(* PLC project Unnamed, Unknown Unnamed 1 *)
(* stored: creationDateTime 2023-03-10T10:37:17, modificationDateTime 2023-03-15T15:56:42 *)

(* ISBN 978-3-8348-0266-8, Lernaufgabe 2.5 *)
FUNCTION_BLOCK Seven_Segment_Display
  VAR_INPUT
    IN0 : BOOL;
    IN1 : BOOL;
    IN2 : BOOL;
    IN3 : BOOL;
    IN4 : BOOL;
  END_VAR
  VAR_OUTPUT
    OUTa : BOOL;
    OUTb : BOOL;
    OUTc : BOOL;
    OUTd : BOOL;
    OUTe : BOOL;
    OUTf : BOOL;
    OUTg : BOOL;
  END_VAR

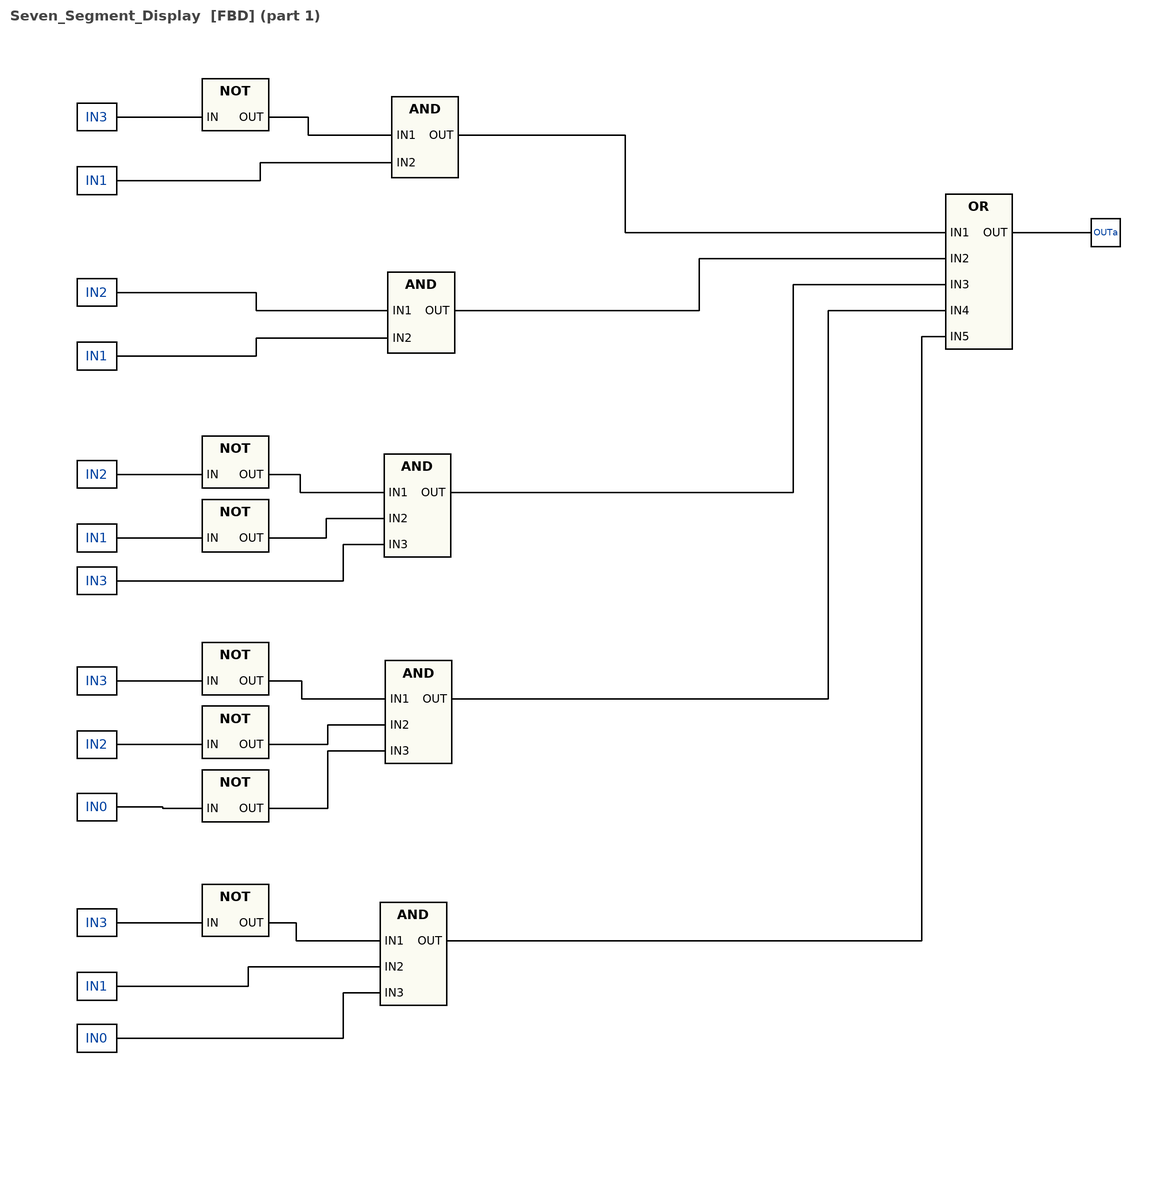
(* FBD diagram, written out as Structured Text *)
OUTa := NOT IN3 AND IN1 OR IN2 AND IN1 OR NOT IN2 AND NOT IN1 AND IN3 OR NOT IN3 AND NOT IN2 AND NOT IN0 OR NOT IN3 AND IN1 AND IN0;
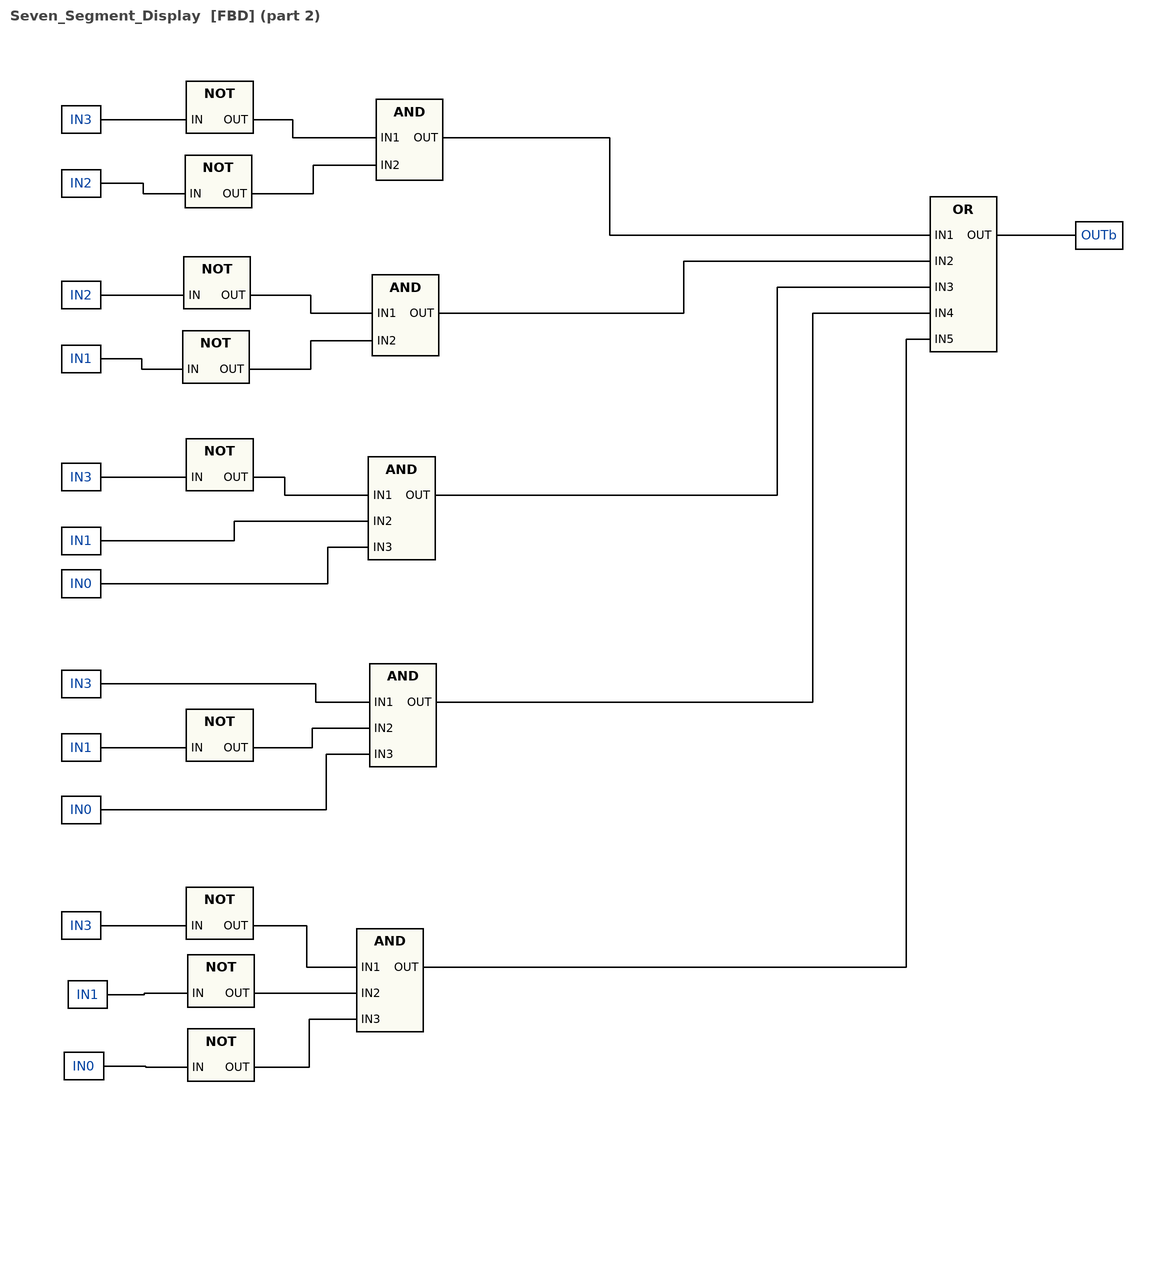
OUTb := NOT IN3 AND NOT IN2 OR NOT IN2 AND NOT IN1 OR NOT IN3 AND IN1 AND IN0 OR IN3 AND NOT IN1 AND IN0 OR NOT IN3 AND NOT IN1 AND NOT IN0;
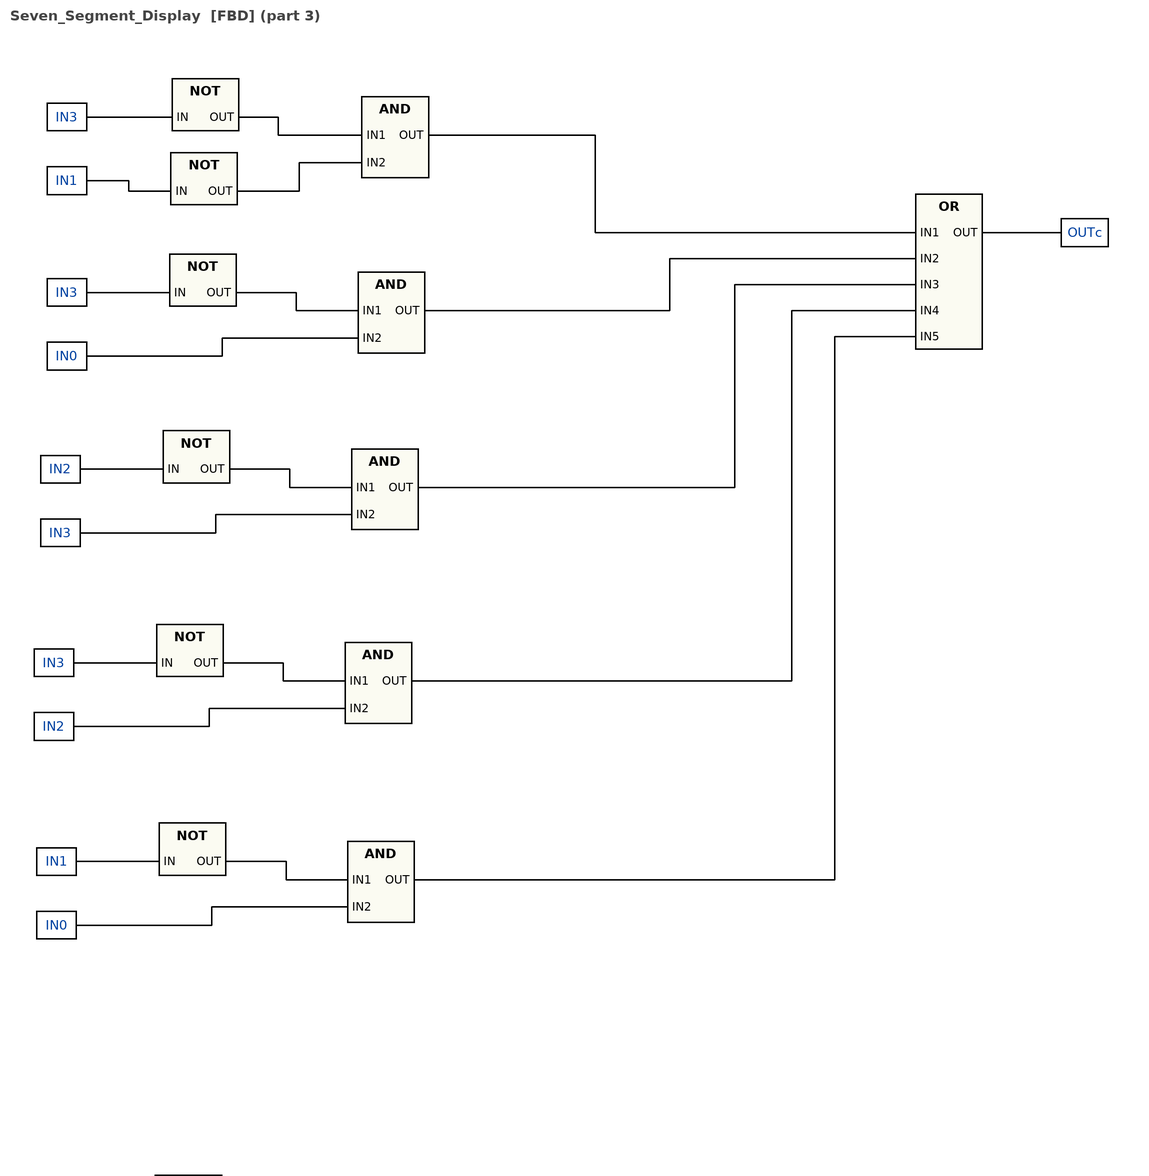
OUTc := NOT IN3 AND NOT IN1 OR NOT IN3 AND IN0 OR NOT IN2 AND IN3 OR NOT IN3 AND IN2 OR NOT IN1 AND IN0;
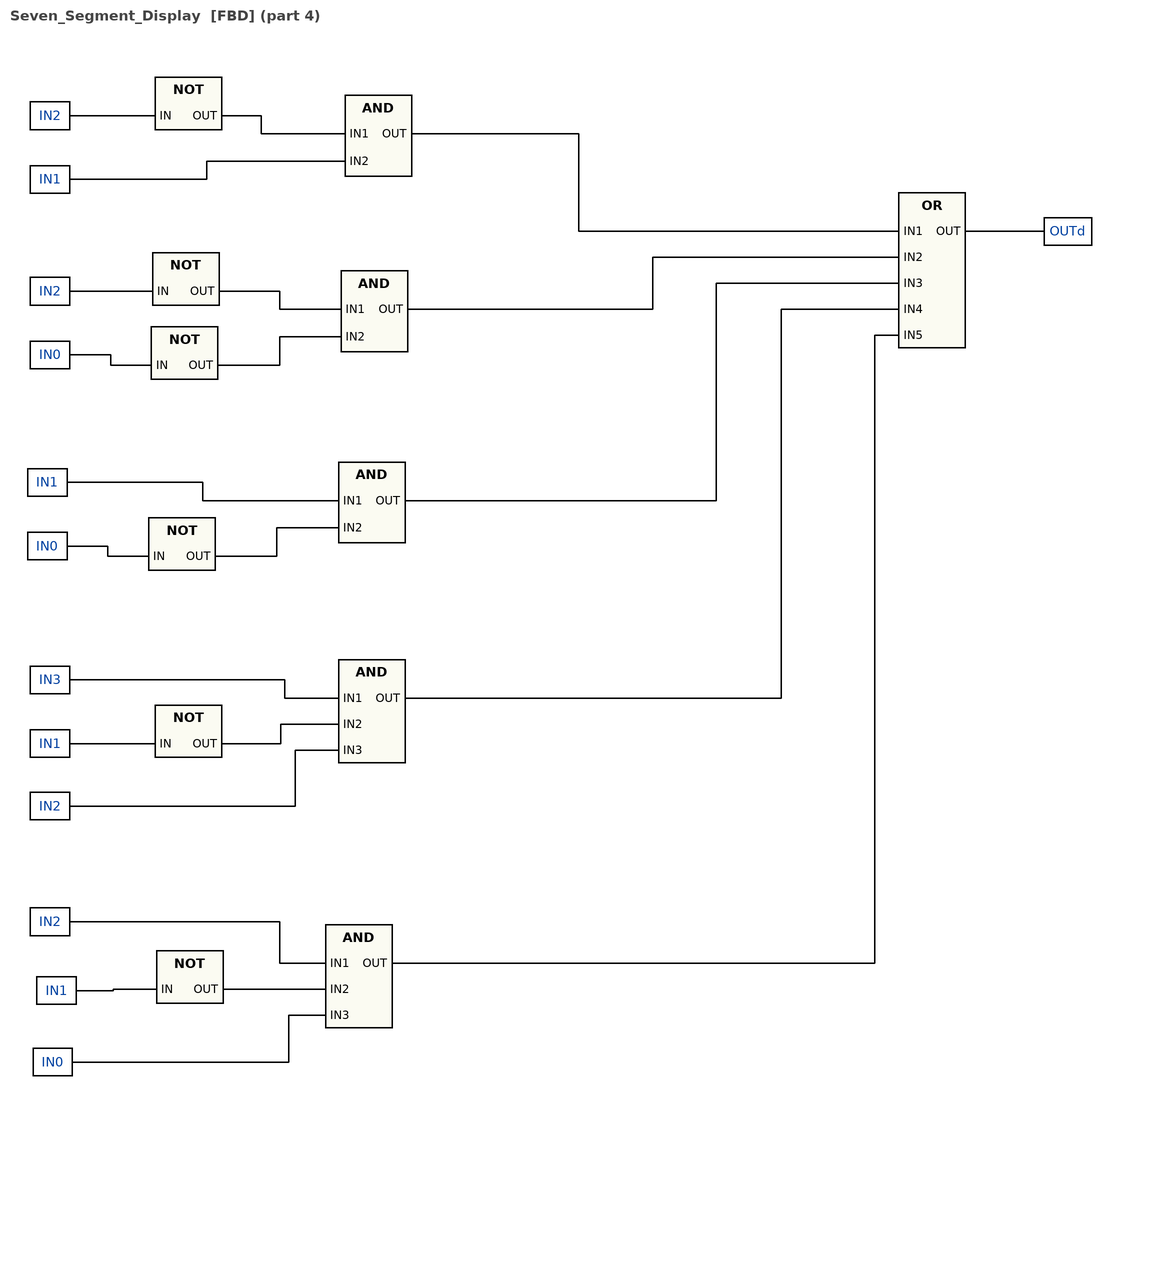
OUTd := NOT IN2 AND IN1 OR NOT IN2 AND NOT IN0 OR IN1 AND NOT IN0 OR IN3 AND NOT IN1 AND IN2 OR IN2 AND NOT IN1 AND IN0;
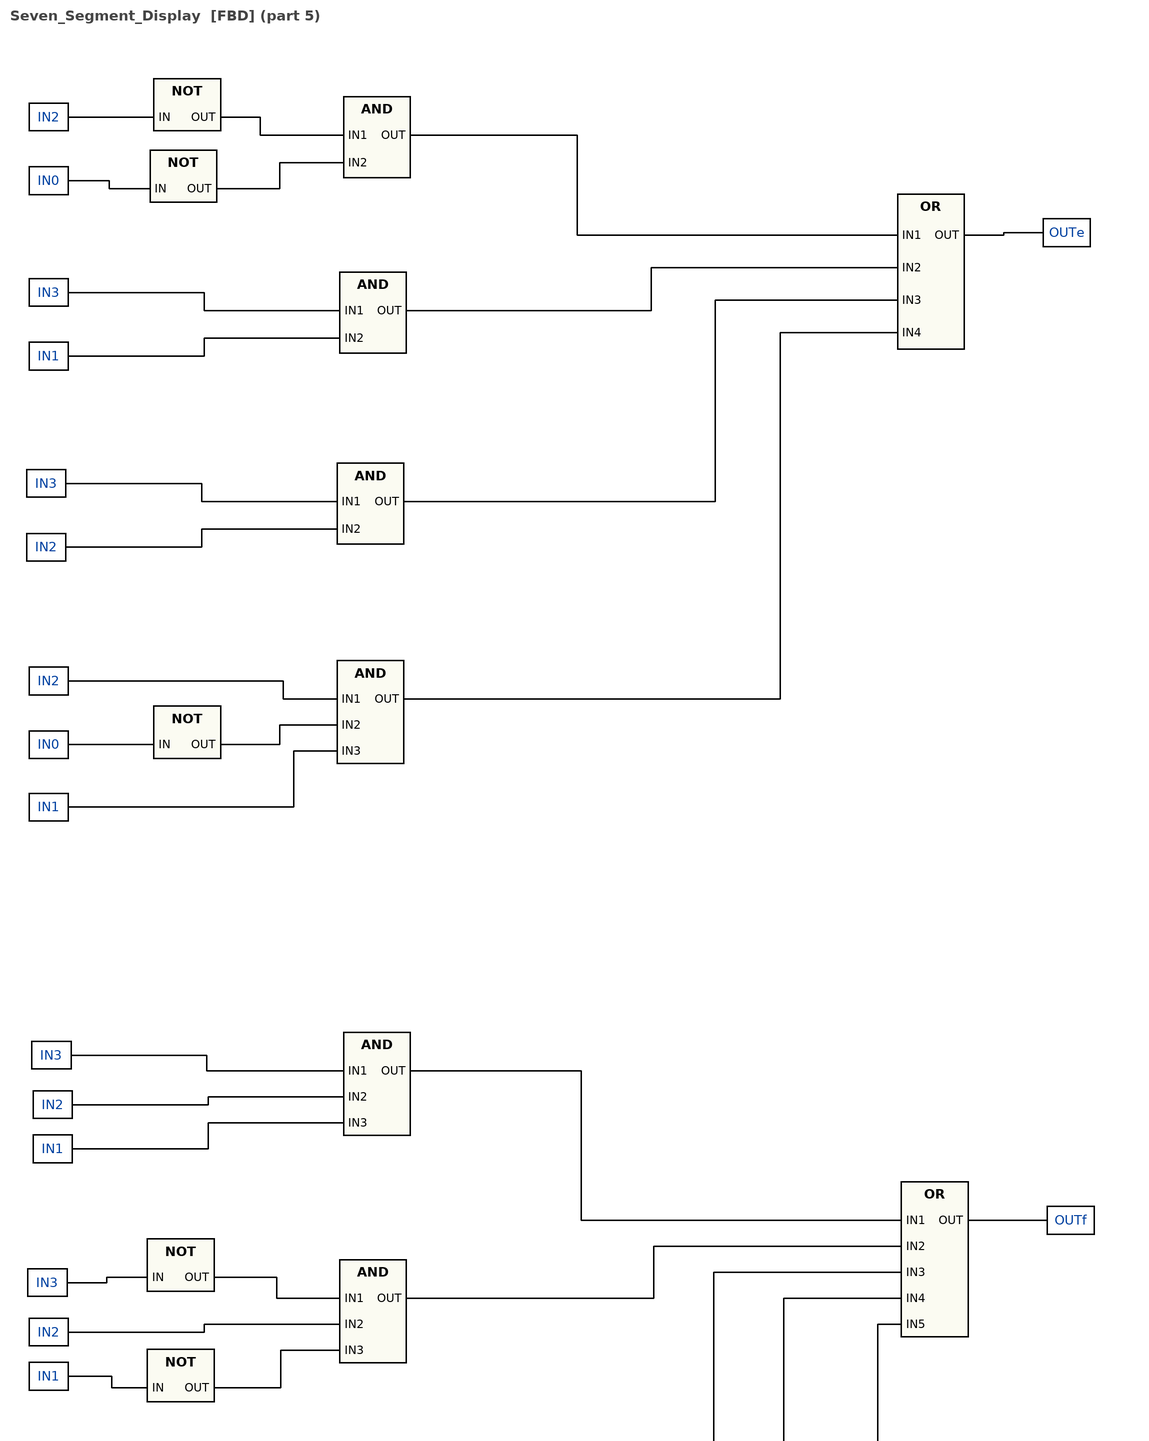
OUTe := NOT IN2 AND NOT IN0 OR IN3 AND IN1 OR IN3 AND IN2 OR IN2 AND NOT IN0 AND IN1;
OUTf := IN3 AND IN2 AND IN1 OR NOT IN3 AND IN2 AND NOT IN1 OR NOT IN3 AND IN2 AND NOT IN0 OR IN3 AND NOT IN2 AND IN0 OR NOT IN2 AND NOT IN1 AND NOT IN0;
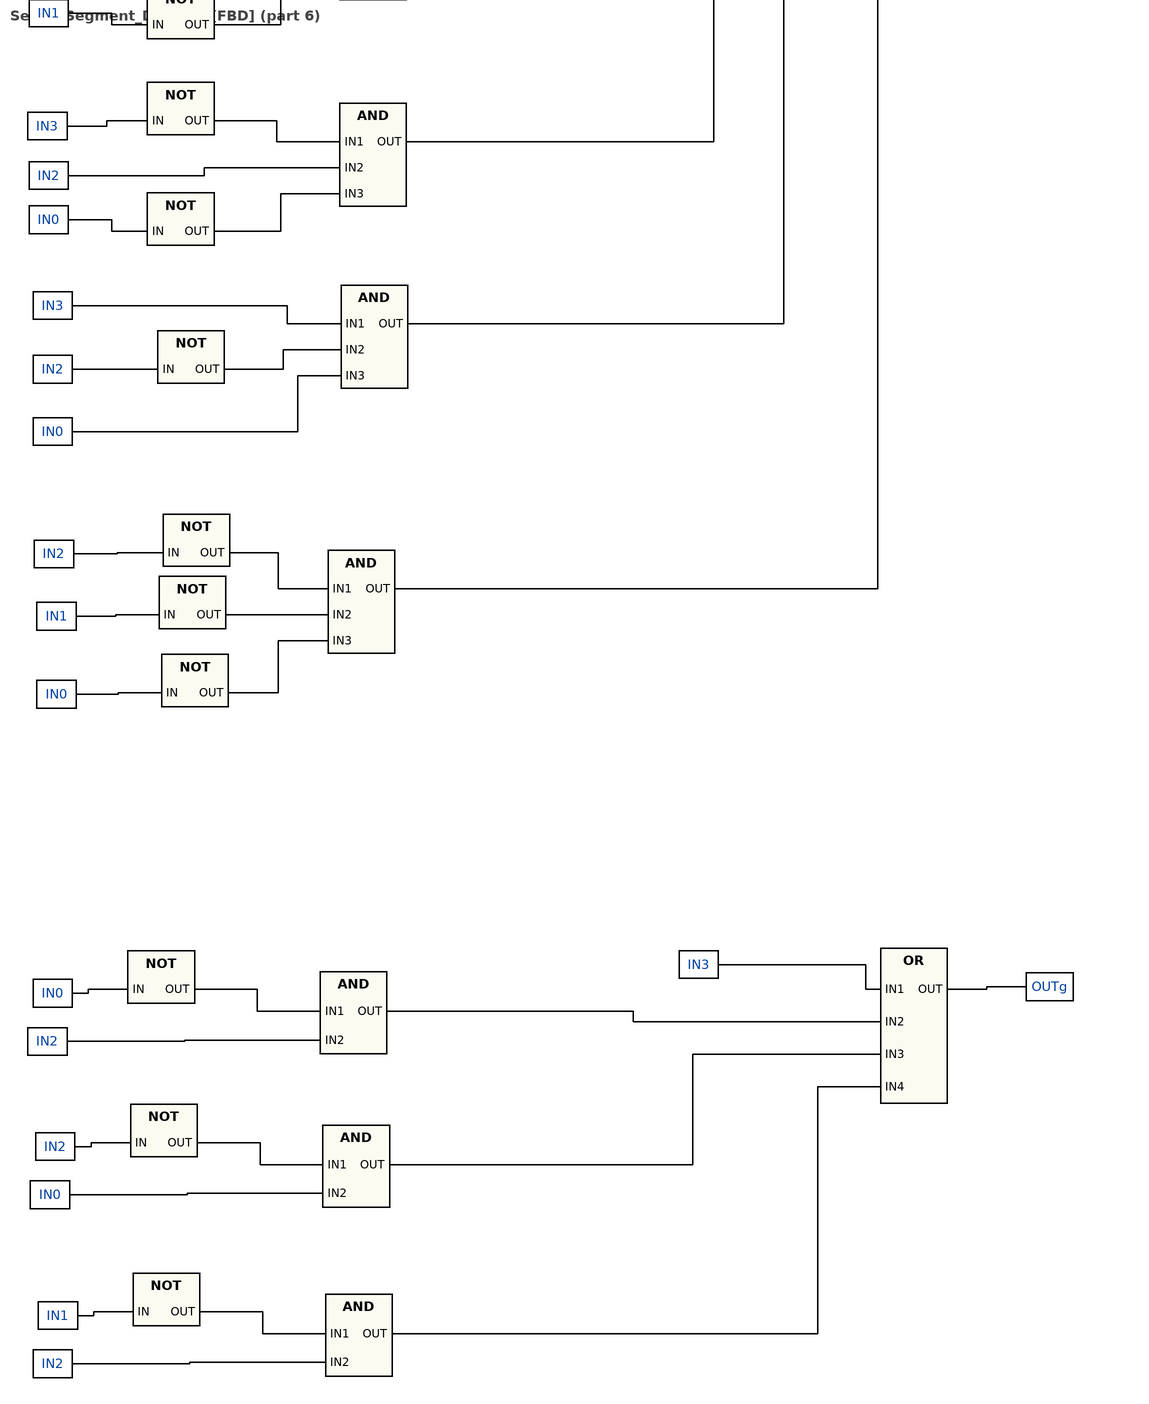
OUTg := IN3 OR NOT IN0 AND IN2 OR NOT IN2 AND IN0 OR NOT IN1 AND IN2;
END_FUNCTION_BLOCK

CONFIGURATION config
  RESOURCE resource1 ON PLC
  END_RESOURCE
END_CONFIGURATION
